        IF finalPosition == 3 THEN
          ;FOLD SPTP P103 Vel=100 % PDAT1 Tool[1]:SMC Base[0] ;%{PE}
          ;FOLD Parameters ;%{h}
          ;Params IlfProvider=kukaroboter.basistech.inlineforms.movement.spline; Kuka.IsGlobalPoint=False; Kuka.PointName=P103; Kuka.BlendingEnabled=False; Kuka.MoveDataPtpName=PDAT1; Kuka.VelocityPtp=100; Kuka.VelocityFieldEnabled=True; Kuka.ColDetectFieldEnabled=True; Kuka.CurrentCDSetIndex=0; Kuka.MovementParameterFieldEnabled=True; IlfCommand=SPTP
          ;ENDFOLD
          SPTP XP103 WITH $VEL_AXIS[1] = SVEL_JOINT(100.0), $TOOL = STOOL2(FP103), $BASE = SBASE(FP103.BASE_NO), $IPO_MODE = SIPO_MODE(FP103.IPO_FRAME), $LOAD = SLOAD(FP103.TOOL_NO), $ACC_AXIS[1] = SACC_JOINT(PPDAT1), $APO = SAPO_PTP(PPDAT1), $GEAR_JERK[1] = SGEAR_JERK(PPDAT1), $COLLMON_TOL_PRO[1] = USE_CM_PRO_VALUES(0)
          ;ENDFOLD
          ;FOLD SLIN P203 Vel=0.1 m/s CPDAT27 Tool[1]:SMC Base[0] ;%{PE}
          ;FOLD Parameters ;%{h}
          ;Params IlfProvider=kukaroboter.basistech.inlineforms.movement.spline; Kuka.IsGlobalPoint=False; Kuka.PointName=P203; Kuka.BlendingEnabled=False; Kuka.MoveDataName=CPDAT27; Kuka.VelocityPath=0.1; Kuka.VelocityFieldEnabled=True; Kuka.ColDetectFieldEnabled=True; Kuka.CurrentCDSetIndex=0; Kuka.MovementParameterFieldEnabled=True; IlfCommand=SLIN
          ;ENDFOLD
          SLIN XP203 WITH $VEL = SVEL_CP(0.1, , LCPDAT27), $TOOL = STOOL2(FP203), $BASE = SBASE(FP203.BASE_NO), $IPO_MODE = SIPO_MODE(FP203.IPO_FRAME), $LOAD = SLOAD(FP203.TOOL_NO), $ACC = SACC_CP(LCPDAT27), $ORI_TYPE = SORI_TYP(LCPDAT27), $APO = SAPO(LCPDAT27), $JERK = SJERK(LCPDAT27), $COLLMON_TOL_PRO[1] = USE_CM_PRO_VALUES(0)
          ;ENDFOLD
          ;FOLD Gripper SET [1]Gripper1 State=[1]ABIERTA Wait 0.2[s] Check with Strategy 1 ;%{PE}
          ;FOLD Parameters Parameters ;%{h}
          ;Params IlfProvider=GripperTech.GripperSet;setgripper=1;setstate=1;setcont=nocont;waittime=0.2;errorstrategy=1
          ;ENDFOLD
          GRPg_SetStateAndCheck(1, 1, 0.2, 1)
          ;ENDFOLD
          ;FOLD SLIN P103 Vel=0.1 m/s CPDAT28 Tool[1]:SMC Base[0] ;%{PE}
          ;FOLD Parameters ;%{h}
          ;Params IlfProvider=kukaroboter.basistech.inlineforms.movement.spline; Kuka.IsGlobalPoint=False; Kuka.PointName=P103; Kuka.BlendingEnabled=False; Kuka.MoveDataName=CPDAT28; Kuka.VelocityPath=0.1; Kuka.VelocityFieldEnabled=True; Kuka.ColDetectFieldEnabled=True; Kuka.CurrentCDSetIndex=0; Kuka.MovementParameterFieldEnabled=True; IlfCommand=SLIN
          ;ENDFOLD
          SLIN XP103 WITH $VEL = SVEL_CP(0.1, , LCPDAT28), $TOOL = STOOL2(FP103), $BASE = SBASE(FP103.BASE_NO), $IPO_MODE = SIPO_MODE(FP103.IPO_FRAME), $LOAD = SLOAD(FP103.TOOL_NO), $ACC = SACC_CP(LCPDAT28), $ORI_TYPE = SORI_TYP(LCPDAT28), $APO = SAPO(LCPDAT28), $JERK = SJERK(LCPDAT28), $COLLMON_TOL_PRO[1] = USE_CM_PRO_VALUES(0)
          ;ENDFOLD
          ;FOLD SPTP P600 Vel=100 % PDAT1 Tool[1]:SMC Base[0] ;%{PE}
          ;FOLD Parameters ;%{h}
          ;Params IlfProvider=kukaroboter.basistech.inlineforms.movement.spline; Kuka.IsGlobalPoint=False; Kuka.PointName=P600; Kuka.BlendingEnabled=False; Kuka.MoveDataPtpName=PDAT1; Kuka.VelocityPtp=100; Kuka.VelocityFieldEnabled=True; Kuka.ColDetectFieldEnabled=True; Kuka.CurrentCDSetIndex=0; Kuka.MovementParameterFieldEnabled=True; IlfCommand=SPTP
          ;ENDFOLD
          SPTP XP600 WITH $VEL_AXIS[1] = SVEL_JOINT(100.0), $TOOL = STOOL2(FP600), $BASE = SBASE(FP600.BASE_NO), $IPO_MODE = SIPO_MODE(FP600.IPO_FRAME), $LOAD = SLOAD(FP600.TOOL_NO), $ACC_AXIS[1] = SACC_JOINT(PPDAT1), $APO = SAPO_PTP(PPDAT1), $GEAR_JERK[1] = SGEAR_JERK(PPDAT1), $COLLMON_TOL_PRO[1] = USE_CM_PRO_VALUES(0)
          ;ENDFOLD
          ;FOLD SLIN P601 Vel=0.1 m/s CPDAT27 Tool[1]:SMC Base[0] ;%{PE}
          ;FOLD Parameters ;%{h}
          ;Params IlfProvider=kukaroboter.basistech.inlineforms.movement.spline; Kuka.IsGlobalPoint=False; Kuka.PointName=P601; Kuka.BlendingEnabled=False; Kuka.MoveDataName=CPDAT27; Kuka.VelocityPath=0.1; Kuka.VelocityFieldEnabled=True; Kuka.ColDetectFieldEnabled=True; Kuka.CurrentCDSetIndex=0; Kuka.MovementParameterFieldEnabled=True; IlfCommand=SLIN
          ;ENDFOLD
          SLIN XP601 WITH $VEL = SVEL_CP(0.1, , LCPDAT27), $TOOL = STOOL2(FP601), $BASE = SBASE(FP601.BASE_NO), $IPO_MODE = SIPO_MODE(FP601.IPO_FRAME), $LOAD = SLOAD(FP601.TOOL_NO), $ACC = SACC_CP(LCPDAT27), $ORI_TYPE = SORI_TYP(LCPDAT27), $APO = SAPO(LCPDAT27), $JERK = SJERK(LCPDAT27), $COLLMON_TOL_PRO[1] = USE_CM_PRO_VALUES(0)
          ;ENDFOLD
          ;FOLD SLIN P602 Vel=0.1 m/s CPDAT27 Tool[1]:SMC Base[0] ;%{PE}
          ;FOLD Parameters ;%{h}
          ;Params IlfProvider=kukaroboter.basistech.inlineforms.movement.spline; Kuka.IsGlobalPoint=False; Kuka.PointName=P602; Kuka.BlendingEnabled=False; Kuka.MoveDataName=CPDAT27; Kuka.VelocityPath=0.1; Kuka.VelocityFieldEnabled=True; Kuka.ColDetectFieldEnabled=True; Kuka.CurrentCDSetIndex=0; Kuka.MovementParameterFieldEnabled=True; IlfCommand=SLIN
          ;ENDFOLD
          SLIN XP602 WITH $VEL = SVEL_CP(0.1, , LCPDAT27), $TOOL = STOOL2(FP602), $BASE = SBASE(FP602.BASE_NO), $IPO_MODE = SIPO_MODE(FP602.IPO_FRAME), $LOAD = SLOAD(FP602.TOOL_NO), $ACC = SACC_CP(LCPDAT27), $ORI_TYPE = SORI_TYP(LCPDAT27), $APO = SAPO(LCPDAT27), $JERK = SJERK(LCPDAT27), $COLLMON_TOL_PRO[1] = USE_CM_PRO_VALUES(0)
          ;ENDFOLD
        ENDIF

        IF finalPosition == 4 THEN
          ;FOLD SPTP P104 Vel=100 % PDAT1 Tool[1]:SMC Base[0] ;%{PE}
          ;FOLD Parameters ;%{h}
          ;Params IlfProvider=kukaroboter.basistech.inlineforms.movement.spline; Kuka.IsGlobalPoint=False; Kuka.PointName=P104; Kuka.BlendingEnabled=False; Kuka.MoveDataPtpName=PDAT1; Kuka.VelocityPtp=100; Kuka.VelocityFieldEnabled=True; Kuka.ColDetectFieldEnabled=True; Kuka.CurrentCDSetIndex=0; Kuka.MovementParameterFieldEnabled=True; IlfCommand=SPTP
          ;ENDFOLD
          SPTP XP104 WITH $VEL_AXIS[1] = SVEL_JOINT(100.0), $TOOL = STOOL2(FP104), $BASE = SBASE(FP104.BASE_NO), $IPO_MODE = SIPO_MODE(FP104.IPO_FRAME), $LOAD = SLOAD(FP104.TOOL_NO), $ACC_AXIS[1] = SACC_JOINT(PPDAT1), $APO = SAPO_PTP(PPDAT1), $GEAR_JERK[1] = SGEAR_JERK(PPDAT1), $COLLMON_TOL_PRO[1] = USE_CM_PRO_VALUES(0)
          ;ENDFOLD
          ;FOLD SLIN P204 Vel=0.1 m/s CPDAT27 Tool[1]:SMC Base[0] ;%{PE}
          ;FOLD Parameters ;%{h}
          ;Params IlfProvider=kukaroboter.basistech.inlineforms.movement.spline; Kuka.IsGlobalPoint=False; Kuka.PointName=P204; Kuka.BlendingEnabled=False; Kuka.MoveDataName=CPDAT27; Kuka.VelocityPath=0.1; Kuka.VelocityFieldEnabled=True; Kuka.ColDetectFieldEnabled=True; Kuka.CurrentCDSetIndex=0; Kuka.MovementParameterFieldEnabled=True; IlfCommand=SLIN
          ;ENDFOLD
          SLIN XP204 WITH $VEL = SVEL_CP(0.1, , LCPDAT27), $TOOL = STOOL2(FP204), $BASE = SBASE(FP204.BASE_NO), $IPO_MODE = SIPO_MODE(FP204.IPO_FRAME), $LOAD = SLOAD(FP204.TOOL_NO), $ACC = SACC_CP(LCPDAT27), $ORI_TYPE = SORI_TYP(LCPDAT27), $APO = SAPO(LCPDAT27), $JERK = SJERK(LCPDAT27), $COLLMON_TOL_PRO[1] = USE_CM_PRO_VALUES(0)
          ;ENDFOLD
          ;FOLD Gripper SET [1]Gripper1 State=[1]ABIERTA Wait 0.2[s] Check with Strategy 1 ;%{PE}
          ;FOLD Parameters Parameters ;%{h}
          ;Params IlfProvider=GripperTech.GripperSet;setgripper=1;setstate=1;setcont=nocont;waittime=0.2;errorstrategy=1
          ;ENDFOLD
          GRPg_SetStateAndCheck(1, 1, 0.2, 1)
          ;ENDFOLD
          ;FOLD SLIN P104 Vel=0.1 m/s CPDAT28 Tool[1]:SMC Base[0] ;%{PE}
          ;FOLD Parameters ;%{h}
          ;Params IlfProvider=kukaroboter.basistech.inlineforms.movement.spline; Kuka.IsGlobalPoint=False; Kuka.PointName=P104; Kuka.BlendingEnabled=False; Kuka.MoveDataName=CPDAT28; Kuka.VelocityPath=0.1; Kuka.VelocityFieldEnabled=True; Kuka.ColDetectFieldEnabled=True; Kuka.CurrentCDSetIndex=0; Kuka.MovementParameterFieldEnabled=True; IlfCommand=SLIN
          ;ENDFOLD
          SLIN XP104 WITH $VEL = SVEL_CP(0.1, , LCPDAT28), $TOOL = STOOL2(FP104), $BASE = SBASE(FP104.BASE_NO), $IPO_MODE = SIPO_MODE(FP104.IPO_FRAME), $LOAD = SLOAD(FP104.TOOL_NO), $ACC = SACC_CP(LCPDAT28), $ORI_TYPE = SORI_TYP(LCPDAT28), $APO = SAPO(LCPDAT28), $JERK = SJERK(LCPDAT28), $COLLMON_TOL_PRO[1] = USE_CM_PRO_VALUES(0)
          ;ENDFOLD
          ;FOLD SPTP P600 Vel=100 % PDAT1 Tool[1]:SMC Base[0] ;%{PE}
          ;FOLD Parameters ;%{h}
          ;Params IlfProvider=kukaroboter.basistech.inlineforms.movement.spline; Kuka.IsGlobalPoint=False; Kuka.PointName=P600; Kuka.BlendingEnabled=False; Kuka.MoveDataPtpName=PDAT1; Kuka.VelocityPtp=100; Kuka.VelocityFieldEnabled=True; Kuka.ColDetectFieldEnabled=True; Kuka.CurrentCDSetIndex=0; Kuka.MovementParameterFieldEnabled=True; IlfCommand=SPTP
          ;ENDFOLD
          SPTP XP600 WITH $VEL_AXIS[1] = SVEL_JOINT(100.0), $TOOL = STOOL2(FP600), $BASE = SBASE(FP600.BASE_NO), $IPO_MODE = SIPO_MODE(FP600.IPO_FRAME), $LOAD = SLOAD(FP600.TOOL_NO), $ACC_AXIS[1] = SACC_JOINT(PPDAT1), $APO = SAPO_PTP(PPDAT1), $GEAR_JERK[1] = SGEAR_JERK(PPDAT1), $COLLMON_TOL_PRO[1] = USE_CM_PRO_VALUES(0)
          ;ENDFOLD
          ;FOLD SLIN P601 Vel=0.1 m/s CPDAT27 Tool[1]:SMC Base[0] ;%{PE}
          ;FOLD Parameters ;%{h}
          ;Params IlfProvider=kukaroboter.basistech.inlineforms.movement.spline; Kuka.IsGlobalPoint=False; Kuka.PointName=P601; Kuka.BlendingEnabled=False; Kuka.MoveDataName=CPDAT27; Kuka.VelocityPath=0.1; Kuka.VelocityFieldEnabled=True; Kuka.ColDetectFieldEnabled=True; Kuka.CurrentCDSetIndex=0; Kuka.MovementParameterFieldEnabled=True; IlfCommand=SLIN
          ;ENDFOLD
          SLIN XP601 WITH $VEL = SVEL_CP(0.1, , LCPDAT27), $TOOL = STOOL2(FP601), $BASE = SBASE(FP601.BASE_NO), $IPO_MODE = SIPO_MODE(FP601.IPO_FRAME), $LOAD = SLOAD(FP601.TOOL_NO), $ACC = SACC_CP(LCPDAT27), $ORI_TYPE = SORI_TYP(LCPDAT27), $APO = SAPO(LCPDAT27), $JERK = SJERK(LCPDAT27), $COLLMON_TOL_PRO[1] = USE_CM_PRO_VALUES(0)
          ;ENDFOLD
          ;FOLD SLIN P602 Vel=0.1 m/s CPDAT27 Tool[1]:SMC Base[0] ;%{PE}
          ;FOLD Parameters ;%{h}
          ;Params IlfProvider=kukaroboter.basistech.inlineforms.movement.spline; Kuka.IsGlobalPoint=False; Kuka.PointName=P602; Kuka.BlendingEnabled=False; Kuka.MoveDataName=CPDAT27; Kuka.VelocityPath=0.1; Kuka.VelocityFieldEnabled=True; Kuka.ColDetectFieldEnabled=True; Kuka.CurrentCDSetIndex=0; Kuka.MovementParameterFieldEnabled=True; IlfCommand=SLIN
          ;ENDFOLD
          SLIN XP602 WITH $VEL = SVEL_CP(0.1, , LCPDAT27), $TOOL = STOOL2(FP602), $BASE = SBASE(FP602.BASE_NO), $IPO_MODE = SIPO_MODE(FP602.IPO_FRAME), $LOAD = SLOAD(FP602.TOOL_NO), $ACC = SACC_CP(LCPDAT27), $ORI_TYPE = SORI_TYP(LCPDAT27), $APO = SAPO(LCPDAT27), $JERK = SJERK(LCPDAT27), $COLLMON_TOL_PRO[1] = USE_CM_PRO_VALUES(0)
          ;ENDFOLD
        ENDIF

        IF finalPosition == 5 THEN
          ;FOLD SPTP P105 Vel=100 % PDAT1 Tool[1]:SMC Base[0] ;%{PE}
          ;FOLD Parameters ;%{h}
          ;Params IlfProvider=kukaroboter.basistech.inlineforms.movement.spline; Kuka.IsGlobalPoint=False; Kuka.PointName=P105; Kuka.BlendingEnabled=False; Kuka.MoveDataPtpName=PDAT1; Kuka.VelocityPtp=100; Kuka.VelocityFieldEnabled=True; Kuka.ColDetectFieldEnabled=True; Kuka.CurrentCDSetIndex=0; Kuka.MovementParameterFieldEnabled=True; IlfCommand=SPTP
          ;ENDFOLD
          SPTP XP105 WITH $VEL_AXIS[1] = SVEL_JOINT(100.0), $TOOL = STOOL2(FP105), $BASE = SBASE(FP105.BASE_NO), $IPO_MODE = SIPO_MODE(FP105.IPO_FRAME), $LOAD = SLOAD(FP105.TOOL_NO), $ACC_AXIS[1] = SACC_JOINT(PPDAT1), $APO = SAPO_PTP(PPDAT1), $GEAR_JERK[1] = SGEAR_JERK(PPDAT1), $COLLMON_TOL_PRO[1] = USE_CM_PRO_VALUES(0)
          ;ENDFOLD
          ;FOLD SLIN P205 Vel=0.1 m/s CPDAT27 Tool[1]:SMC Base[0] ;%{PE}
          ;FOLD Parameters ;%{h}
          ;Params IlfProvider=kukaroboter.basistech.inlineforms.movement.spline; Kuka.IsGlobalPoint=False; Kuka.PointName=P205; Kuka.BlendingEnabled=False; Kuka.MoveDataName=CPDAT27; Kuka.VelocityPath=0.1; Kuka.VelocityFieldEnabled=True; Kuka.ColDetectFieldEnabled=True; Kuka.CurrentCDSetIndex=0; Kuka.MovementParameterFieldEnabled=True; IlfCommand=SLIN
          ;ENDFOLD
          SLIN XP205 WITH $VEL = SVEL_CP(0.1, , LCPDAT27), $TOOL = STOOL2(FP205), $BASE = SBASE(FP205.BASE_NO), $IPO_MODE = SIPO_MODE(FP205.IPO_FRAME), $LOAD = SLOAD(FP205.TOOL_NO), $ACC = SACC_CP(LCPDAT27), $ORI_TYPE = SORI_TYP(LCPDAT27), $APO = SAPO(LCPDAT27), $JERK = SJERK(LCPDAT27), $COLLMON_TOL_PRO[1] = USE_CM_PRO_VALUES(0)
          ;ENDFOLD
          ;FOLD Gripper SET [1]Gripper1 State=[1]ABIERTA Wait 0.2[s] Check with Strategy 1 ;%{PE}
          ;FOLD Parameters Parameters ;%{h}
          ;Params IlfProvider=GripperTech.GripperSet;setgripper=1;setstate=1;setcont=nocont;waittime=0.2;errorstrategy=1
          ;ENDFOLD
          GRPg_SetStateAndCheck(1, 1, 0.2, 1)
          ;ENDFOLD
          ;FOLD SLIN P105 Vel=0.1 m/s CPDAT28 Tool[1]:SMC Base[0] ;%{PE}
          ;FOLD Parameters ;%{h}
          ;Params IlfProvider=kukaroboter.basistech.inlineforms.movement.spline; Kuka.IsGlobalPoint=False; Kuka.PointName=P105; Kuka.BlendingEnabled=False; Kuka.MoveDataName=CPDAT28; Kuka.VelocityPath=0.1; Kuka.VelocityFieldEnabled=True; Kuka.ColDetectFieldEnabled=True; Kuka.CurrentCDSetIndex=0; Kuka.MovementParameterFieldEnabled=True; IlfCommand=SLIN
          ;ENDFOLD
          SLIN XP105 WITH $VEL = SVEL_CP(0.1, , LCPDAT28), $TOOL = STOOL2(FP105), $BASE = SBASE(FP105.BASE_NO), $IPO_MODE = SIPO_MODE(FP105.IPO_FRAME), $LOAD = SLOAD(FP105.TOOL_NO), $ACC = SACC_CP(LCPDAT28), $ORI_TYPE = SORI_TYP(LCPDAT28), $APO = SAPO(LCPDAT28), $JERK = SJERK(LCPDAT28), $COLLMON_TOL_PRO[1] = USE_CM_PRO_VALUES(0)
          ;ENDFOLD
          ;FOLD SPTP P600 Vel=100 % PDAT1 Tool[1]:SMC Base[0] ;%{PE}
          ;FOLD Parameters ;%{h}
          ;Params IlfProvider=kukaroboter.basistech.inlineforms.movement.spline; Kuka.IsGlobalPoint=False; Kuka.PointName=P600; Kuka.BlendingEnabled=False; Kuka.MoveDataPtpName=PDAT1; Kuka.VelocityPtp=100; Kuka.VelocityFieldEnabled=True; Kuka.ColDetectFieldEnabled=True; Kuka.CurrentCDSetIndex=0; Kuka.MovementParameterFieldEnabled=True; IlfCommand=SPTP
          ;ENDFOLD
          SPTP XP600 WITH $VEL_AXIS[1] = SVEL_JOINT(100.0), $TOOL = STOOL2(FP600), $BASE = SBASE(FP600.BASE_NO), $IPO_MODE = SIPO_MODE(FP600.IPO_FRAME), $LOAD = SLOAD(FP600.TOOL_NO), $ACC_AXIS[1] = SACC_JOINT(PPDAT1), $APO = SAPO_PTP(PPDAT1), $GEAR_JERK[1] = SGEAR_JERK(PPDAT1), $COLLMON_TOL_PRO[1] = USE_CM_PRO_VALUES(0)
          ;ENDFOLD
          ;FOLD SLIN P601 Vel=0.1 m/s CPDAT27 Tool[1]:SMC Base[0] ;%{PE}
          ;FOLD Parameters ;%{h}
          ;Params IlfProvider=kukaroboter.basistech.inlineforms.movement.spline; Kuka.IsGlobalPoint=False; Kuka.PointName=P601; Kuka.BlendingEnabled=False; Kuka.MoveDataName=CPDAT27; Kuka.VelocityPath=0.1; Kuka.VelocityFieldEnabled=True; Kuka.ColDetectFieldEnabled=True; Kuka.CurrentCDSetIndex=0; Kuka.MovementParameterFieldEnabled=True; IlfCommand=SLIN
          ;ENDFOLD
          SLIN XP601 WITH $VEL = SVEL_CP(0.1, , LCPDAT27), $TOOL = STOOL2(FP601), $BASE = SBASE(FP601.BASE_NO), $IPO_MODE = SIPO_MODE(FP601.IPO_FRAME), $LOAD = SLOAD(FP601.TOOL_NO), $ACC = SACC_CP(LCPDAT27), $ORI_TYPE = SORI_TYP(LCPDAT27), $APO = SAPO(LCPDAT27), $JERK = SJERK(LCPDAT27), $COLLMON_TOL_PRO[1] = USE_CM_PRO_VALUES(0)
          ;ENDFOLD
          ;FOLD SLIN P602 Vel=0.1 m/s CPDAT27 Tool[1]:SMC Base[0] ;%{PE}
          ;FOLD Parameters ;%{h}
          ;Params IlfProvider=kukaroboter.basistech.inlineforms.movement.spline; Kuka.IsGlobalPoint=False; Kuka.PointName=P602; Kuka.BlendingEnabled=False; Kuka.MoveDataName=CPDAT27; Kuka.VelocityPath=0.1; Kuka.VelocityFieldEnabled=True; Kuka.ColDetectFieldEnabled=True; Kuka.CurrentCDSetIndex=0; Kuka.MovementParameterFieldEnabled=True; IlfCommand=SLIN
          ;ENDFOLD
          SLIN XP602 WITH $VEL = SVEL_CP(0.1, , LCPDAT27), $TOOL = STOOL2(FP602), $BASE = SBASE(FP602.BASE_NO), $IPO_MODE = SIPO_MODE(FP602.IPO_FRAME), $LOAD = SLOAD(FP602.TOOL_NO), $ACC = SACC_CP(LCPDAT27), $ORI_TYPE = SORI_TYP(LCPDAT27), $APO = SAPO(LCPDAT27), $JERK = SJERK(LCPDAT27), $COLLMON_TOL_PRO[1] = USE_CM_PRO_VALUES(0)
          ;ENDFOLD
        ENDIF

        IF finalPosition == 6 THEN
          ;FOLD SPTP P106 Vel=100 % PDAT1 Tool[1]:SMC Base[0] ;%{PE}
          ;FOLD Parameters ;%{h}
          ;Params IlfProvider=kukaroboter.basistech.inlineforms.movement.spline; Kuka.IsGlobalPoint=False; Kuka.PointName=P106; Kuka.BlendingEnabled=False; Kuka.MoveDataPtpName=PDAT1; Kuka.VelocityPtp=100; Kuka.VelocityFieldEnabled=True; Kuka.ColDetectFieldEnabled=True; Kuka.CurrentCDSetIndex=0; Kuka.MovementParameterFieldEnabled=True; IlfCommand=SPTP
          ;ENDFOLD
          SPTP XP106 WITH $VEL_AXIS[1] = SVEL_JOINT(100.0), $TOOL = STOOL2(FP106), $BASE = SBASE(FP106.BASE_NO), $IPO_MODE = SIPO_MODE(FP106.IPO_FRAME), $LOAD = SLOAD(FP106.TOOL_NO), $ACC_AXIS[1] = SACC_JOINT(PPDAT1), $APO = SAPO_PTP(PPDAT1), $GEAR_JERK[1] = SGEAR_JERK(PPDAT1), $COLLMON_TOL_PRO[1] = USE_CM_PRO_VALUES(0)
          ;ENDFOLD
          ;FOLD SLIN P206 Vel=0.1 m/s CPDAT27 Tool[1]:SMC Base[0] ;%{PE}
          ;FOLD Parameters ;%{h}
          ;Params IlfProvider=kukaroboter.basistech.inlineforms.movement.spline; Kuka.IsGlobalPoint=False; Kuka.PointName=P206; Kuka.BlendingEnabled=False; Kuka.MoveDataName=CPDAT27; Kuka.VelocityPath=0.1; Kuka.VelocityFieldEnabled=True; Kuka.ColDetectFieldEnabled=True; Kuka.CurrentCDSetIndex=0; Kuka.MovementParameterFieldEnabled=True; IlfCommand=SLIN
          ;ENDFOLD
          SLIN XP206 WITH $VEL = SVEL_CP(0.1, , LCPDAT27), $TOOL = STOOL2(FP206), $BASE = SBASE(FP206.BASE_NO), $IPO_MODE = SIPO_MODE(FP206.IPO_FRAME), $LOAD = SLOAD(FP206.TOOL_NO), $ACC = SACC_CP(LCPDAT27), $ORI_TYPE = SORI_TYP(LCPDAT27), $APO = SAPO(LCPDAT27), $JERK = SJERK(LCPDAT27), $COLLMON_TOL_PRO[1] = USE_CM_PRO_VALUES(0)
          ;ENDFOLD
          ;FOLD Gripper SET [1]Gripper1 State=[1]ABIERTA Wait 0.2[s] Check with Strategy 1 ;%{PE}
          ;FOLD Parameters Parameters ;%{h}
          ;Params IlfProvider=GripperTech.GripperSet;setgripper=1;setstate=1;setcont=nocont;waittime=0.2;errorstrategy=1
          ;ENDFOLD
          GRPg_SetStateAndCheck(1, 1, 0.2, 1)
          ;ENDFOLD
          ;FOLD SLIN P106 Vel=0.1 m/s CPDAT28 Tool[1]:SMC Base[0] ;%{PE}
          ;FOLD Parameters ;%{h}
          ;Params IlfProvider=kukaroboter.basistech.inlineforms.movement.spline; Kuka.IsGlobalPoint=False; Kuka.PointName=P106; Kuka.BlendingEnabled=False; Kuka.MoveDataName=CPDAT28; Kuka.VelocityPath=0.1; Kuka.VelocityFieldEnabled=True; Kuka.ColDetectFieldEnabled=True; Kuka.CurrentCDSetIndex=0; Kuka.MovementParameterFieldEnabled=True; IlfCommand=SLIN
          ;ENDFOLD
          SLIN XP106 WITH $VEL = SVEL_CP(0.1, , LCPDAT28), $TOOL = STOOL2(FP106), $BASE = SBASE(FP106.BASE_NO), $IPO_MODE = SIPO_MODE(FP106.IPO_FRAME), $LOAD = SLOAD(FP106.TOOL_NO), $ACC = SACC_CP(LCPDAT28), $ORI_TYPE = SORI_TYP(LCPDAT28), $APO = SAPO(LCPDAT28), $JERK = SJERK(LCPDAT28), $COLLMON_TOL_PRO[1] = USE_CM_PRO_VALUES(0)
          ;ENDFOLD
          ;FOLD SPTP P600 Vel=100 % PDAT1 Tool[1]:SMC Base[0] ;%{PE}
          ;FOLD Parameters ;%{h}
          ;Params IlfProvider=kukaroboter.basistech.inlineforms.movement.spline; Kuka.IsGlobalPoint=False; Kuka.PointName=P600; Kuka.BlendingEnabled=False; Kuka.MoveDataPtpName=PDAT1; Kuka.VelocityPtp=100; Kuka.VelocityFieldEnabled=True; Kuka.ColDetectFieldEnabled=True; Kuka.CurrentCDSetIndex=0; Kuka.MovementParameterFieldEnabled=True; IlfCommand=SPTP
          ;ENDFOLD
          SPTP XP600 WITH $VEL_AXIS[1] = SVEL_JOINT(100.0), $TOOL = STOOL2(FP600), $BASE = SBASE(FP600.BASE_NO), $IPO_MODE = SIPO_MODE(FP600.IPO_FRAME), $LOAD = SLOAD(FP600.TOOL_NO), $ACC_AXIS[1] = SACC_JOINT(PPDAT1), $APO = SAPO_PTP(PPDAT1), $GEAR_JERK[1] = SGEAR_JERK(PPDAT1), $COLLMON_TOL_PRO[1] = USE_CM_PRO_VALUES(0)
          ;ENDFOLD
          ;FOLD SLIN P601 Vel=0.1 m/s CPDAT27 Tool[1]:SMC Base[0] ;%{PE}
          ;FOLD Parameters ;%{h}
          ;Params IlfProvider=kukaroboter.basistech.inlineforms.movement.spline; Kuka.IsGlobalPoint=False; Kuka.PointName=P601; Kuka.BlendingEnabled=False; Kuka.MoveDataName=CPDAT27; Kuka.VelocityPath=0.1; Kuka.VelocityFieldEnabled=True; Kuka.ColDetectFieldEnabled=True; Kuka.CurrentCDSetIndex=0; Kuka.MovementParameterFieldEnabled=True; IlfCommand=SLIN
          ;ENDFOLD
          SLIN XP601 WITH $VEL = SVEL_CP(0.1, , LCPDAT27), $TOOL = STOOL2(FP601), $BASE = SBASE(FP601.BASE_NO), $IPO_MODE = SIPO_MODE(FP601.IPO_FRAME), $LOAD = SLOAD(FP601.TOOL_NO), $ACC = SACC_CP(LCPDAT27), $ORI_TYPE = SORI_TYP(LCPDAT27), $APO = SAPO(LCPDAT27), $JERK = SJERK(LCPDAT27), $COLLMON_TOL_PRO[1] = USE_CM_PRO_VALUES(0)
          ;ENDFOLD
          ;FOLD SLIN P602 Vel=0.1 m/s CPDAT27 Tool[1]:SMC Base[0] ;%{PE}
          ;FOLD Parameters ;%{h}
          ;Params IlfProvider=kukaroboter.basistech.inlineforms.movement.spline; Kuka.IsGlobalPoint=False; Kuka.PointName=P602; Kuka.BlendingEnabled=False; Kuka.MoveDataName=CPDAT27; Kuka.VelocityPath=0.1; Kuka.VelocityFieldEnabled=True; Kuka.ColDetectFieldEnabled=True; Kuka.CurrentCDSetIndex=0; Kuka.MovementParameterFieldEnabled=True; IlfCommand=SLIN
          ;ENDFOLD
          SLIN XP602 WITH $VEL = SVEL_CP(0.1, , LCPDAT27), $TOOL = STOOL2(FP602), $BASE = SBASE(FP602.BASE_NO), $IPO_MODE = SIPO_MODE(FP602.IPO_FRAME), $LOAD = SLOAD(FP602.TOOL_NO), $ACC = SACC_CP(LCPDAT27), $ORI_TYPE = SORI_TYP(LCPDAT27), $APO = SAPO(LCPDAT27), $JERK = SJERK(LCPDAT27), $COLLMON_TOL_PRO[1] = USE_CM_PRO_VALUES(0)
          ;ENDFOLD
        ENDIF

        IF finalPosition == 7 THEN
          ;FOLD SPTP P107 Vel=100 % PDAT1 Tool[1]:SMC Base[0] ;%{PE}
          ;FOLD Parameters ;%{h}
          ;Params IlfProvider=kukaroboter.basistech.inlineforms.movement.spline; Kuka.IsGlobalPoint=False; Kuka.PointName=P107; Kuka.BlendingEnabled=False; Kuka.MoveDataPtpName=PDAT1; Kuka.VelocityPtp=100; Kuka.VelocityFieldEnabled=True; Kuka.ColDetectFieldEnabled=True; Kuka.CurrentCDSetIndex=0; Kuka.MovementParameterFieldEnabled=True; IlfCommand=SPTP
          ;ENDFOLD
          SPTP XP107 WITH $VEL_AXIS[1] = SVEL_JOINT(100.0), $TOOL = STOOL2(FP107), $BASE = SBASE(FP107.BASE_NO), $IPO_MODE = SIPO_MODE(FP107.IPO_FRAME), $LOAD = SLOAD(FP107.TOOL_NO), $ACC_AXIS[1] = SACC_JOINT(PPDAT1), $APO = SAPO_PTP(PPDAT1), $GEAR_JERK[1] = SGEAR_JERK(PPDAT1), $COLLMON_TOL_PRO[1] = USE_CM_PRO_VALUES(0)
          ;ENDFOLD
          ;FOLD SLIN P207 Vel=0.1 m/s CPDAT27 Tool[1]:SMC Base[0] ;%{PE}
          ;FOLD Parameters ;%{h}
          ;Params IlfProvider=kukaroboter.basistech.inlineforms.movement.spline; Kuka.IsGlobalPoint=False; Kuka.PointName=P207; Kuka.BlendingEnabled=False; Kuka.MoveDataName=CPDAT27; Kuka.VelocityPath=0.1; Kuka.VelocityFieldEnabled=True; Kuka.ColDetectFieldEnabled=True; Kuka.CurrentCDSetIndex=0; Kuka.MovementParameterFieldEnabled=True; IlfCommand=SLIN
          ;ENDFOLD
          SLIN XP207 WITH $VEL = SVEL_CP(0.1, , LCPDAT27), $TOOL = STOOL2(FP207), $BASE = SBASE(FP207.BASE_NO), $IPO_MODE = SIPO_MODE(FP207.IPO_FRAME), $LOAD = SLOAD(FP207.TOOL_NO), $ACC = SACC_CP(LCPDAT27), $ORI_TYPE = SORI_TYP(LCPDAT27), $APO = SAPO(LCPDAT27), $JERK = SJERK(LCPDAT27), $COLLMON_TOL_PRO[1] = USE_CM_PRO_VALUES(0)
          ;ENDFOLD
          ;FOLD Gripper SET [1]Gripper1 State=[1]ABIERTA Wait 0.2[s] Check with Strategy 1 ;%{PE}
          ;FOLD Parameters Parameters ;%{h}
          ;Params IlfProvider=GripperTech.GripperSet;setgripper=1;setstate=1;setcont=nocont;waittime=0.2;errorstrategy=1
          ;ENDFOLD
          GRPg_SetStateAndCheck(1, 1, 0.2, 1)
          ;ENDFOLD
          ;FOLD SLIN P107 Vel=0.1 m/s CPDAT28 Tool[1]:SMC Base[0] ;%{PE}
          ;FOLD Parameters ;%{h}
          ;Params IlfProvider=kukaroboter.basistech.inlineforms.movement.spline; Kuka.IsGlobalPoint=False; Kuka.PointName=P107; Kuka.BlendingEnabled=False; Kuka.MoveDataName=CPDAT28; Kuka.VelocityPath=0.1; Kuka.VelocityFieldEnabled=True; Kuka.ColDetectFieldEnabled=True; Kuka.CurrentCDSetIndex=0; Kuka.MovementParameterFieldEnabled=True; IlfCommand=SLIN
          ;ENDFOLD
          SLIN XP107 WITH $VEL = SVEL_CP(0.1, , LCPDAT28), $TOOL = STOOL2(FP107), $BASE = SBASE(FP107.BASE_NO), $IPO_MODE = SIPO_MODE(FP107.IPO_FRAME), $LOAD = SLOAD(FP107.TOOL_NO), $ACC = SACC_CP(LCPDAT28), $ORI_TYPE = SORI_TYP(LCPDAT28), $APO = SAPO(LCPDAT28), $JERK = SJERK(LCPDAT28), $COLLMON_TOL_PRO[1] = USE_CM_PRO_VALUES(0)
          ;ENDFOLD
          ;FOLD SPTP P600 Vel=100 % PDAT1 Tool[1]:SMC Base[0] ;%{PE}
          ;FOLD Parameters ;%{h}
          ;Params IlfProvider=kukaroboter.basistech.inlineforms.movement.spline; Kuka.IsGlobalPoint=False; Kuka.PointName=P600; Kuka.BlendingEnabled=False; Kuka.MoveDataPtpName=PDAT1; Kuka.VelocityPtp=100; Kuka.VelocityFieldEnabled=True; Kuka.ColDetectFieldEnabled=True; Kuka.CurrentCDSetIndex=0; Kuka.MovementParameterFieldEnabled=True; IlfCommand=SPTP
          ;ENDFOLD
          SPTP XP600 WITH $VEL_AXIS[1] = SVEL_JOINT(100.0), $TOOL = STOOL2(FP600), $BASE = SBASE(FP600.BASE_NO), $IPO_MODE = SIPO_MODE(FP600.IPO_FRAME), $LOAD = SLOAD(FP600.TOOL_NO), $ACC_AXIS[1] = SACC_JOINT(PPDAT1), $APO = SAPO_PTP(PPDAT1), $GEAR_JERK[1] = SGEAR_JERK(PPDAT1), $COLLMON_TOL_PRO[1] = USE_CM_PRO_VALUES(0)
          ;ENDFOLD
          ;FOLD SLIN P601 Vel=0.1 m/s CPDAT27 Tool[1]:SMC Base[0] ;%{PE}
          ;FOLD Parameters ;%{h}
          ;Params IlfProvider=kukaroboter.basistech.inlineforms.movement.spline; Kuka.IsGlobalPoint=False; Kuka.PointName=P601; Kuka.BlendingEnabled=False; Kuka.MoveDataName=CPDAT27; Kuka.VelocityPath=0.1; Kuka.VelocityFieldEnabled=True; Kuka.ColDetectFieldEnabled=True; Kuka.CurrentCDSetIndex=0; Kuka.MovementParameterFieldEnabled=True; IlfCommand=SLIN
          ;ENDFOLD
          SLIN XP601 WITH $VEL = SVEL_CP(0.1, , LCPDAT27), $TOOL = STOOL2(FP601), $BASE = SBASE(FP601.BASE_NO), $IPO_MODE = SIPO_MODE(FP601.IPO_FRAME), $LOAD = SLOAD(FP601.TOOL_NO), $ACC = SACC_CP(LCPDAT27), $ORI_TYPE = SORI_TYP(LCPDAT27), $APO = SAPO(LCPDAT27), $JERK = SJERK(LCPDAT27), $COLLMON_TOL_PRO[1] = USE_CM_PRO_VALUES(0)
          ;ENDFOLD
          ;FOLD SLIN P602 Vel=0.1 m/s CPDAT27 Tool[1]:SMC Base[0] ;%{PE}
          ;FOLD Parameters ;%{h}
          ;Params IlfProvider=kukaroboter.basistech.inlineforms.movement.spline; Kuka.IsGlobalPoint=False; Kuka.PointName=P602; Kuka.BlendingEnabled=False; Kuka.MoveDataName=CPDAT27; Kuka.VelocityPath=0.1; Kuka.VelocityFieldEnabled=True; Kuka.ColDetectFieldEnabled=True; Kuka.CurrentCDSetIndex=0; Kuka.MovementParameterFieldEnabled=True; IlfCommand=SLIN
          ;ENDFOLD
          SLIN XP602 WITH $VEL = SVEL_CP(0.1, , LCPDAT27), $TOOL = STOOL2(FP602), $BASE = SBASE(FP602.BASE_NO), $IPO_MODE = SIPO_MODE(FP602.IPO_FRAME), $LOAD = SLOAD(FP602.TOOL_NO), $ACC = SACC_CP(LCPDAT27), $ORI_TYPE = SORI_TYP(LCPDAT27), $APO = SAPO(LCPDAT27), $JERK = SJERK(LCPDAT27), $COLLMON_TOL_PRO[1] = USE_CM_PRO_VALUES(0)
          ;ENDFOLD
        ENDIF

        IF finalPosition == 8 THEN
          ;FOLD SPTP P108 Vel=100 % PDAT1 Tool[1]:SMC Base[0] ;%{PE}
          ;FOLD Parameters ;%{h}
          ;Params IlfProvider=kukaroboter.basistech.inlineforms.movement.spline; Kuka.IsGlobalPoint=False; Kuka.PointName=P108; Kuka.BlendingEnabled=False; Kuka.MoveDataPtpName=PDAT1; Kuka.VelocityPtp=100; Kuka.VelocityFieldEnabled=True; Kuka.ColDetectFieldEnabled=True; Kuka.CurrentCDSetIndex=0; Kuka.MovementParameterFieldEnabled=True; IlfCommand=SPTP
          ;ENDFOLD
          SPTP XP108 WITH $VEL_AXIS[1] = SVEL_JOINT(100.0), $TOOL = STOOL2(FP108), $BASE = SBASE(FP108.BASE_NO), $IPO_MODE = SIPO_MODE(FP108.IPO_FRAME), $LOAD = SLOAD(FP108.TOOL_NO), $ACC_AXIS[1] = SACC_JOINT(PPDAT1), $APO = SAPO_PTP(PPDAT1), $GEAR_JERK[1] = SGEAR_JERK(PPDAT1), $COLLMON_TOL_PRO[1] = USE_CM_PRO_VALUES(0)
          ;ENDFOLD
          ;FOLD SLIN P208 Vel=0.1 m/s CPDAT27 Tool[1]:SMC Base[0] ;%{PE}
          ;FOLD Parameters ;%{h}
          ;Params IlfProvider=kukaroboter.basistech.inlineforms.movement.spline; Kuka.IsGlobalPoint=False; Kuka.PointName=P208; Kuka.BlendingEnabled=False; Kuka.MoveDataName=CPDAT27; Kuka.VelocityPath=0.1; Kuka.VelocityFieldEnabled=True; Kuka.ColDetectFieldEnabled=True; Kuka.CurrentCDSetIndex=0; Kuka.MovementParameterFieldEnabled=True; IlfCommand=SLIN
          ;ENDFOLD
          SLIN XP208 WITH $VEL = SVEL_CP(0.1, , LCPDAT27), $TOOL = STOOL2(FP208), $BASE = SBASE(FP208.BASE_NO), $IPO_MODE = SIPO_MODE(FP208.IPO_FRAME), $LOAD = SLOAD(FP208.TOOL_NO), $ACC = SACC_CP(LCPDAT27), $ORI_TYPE = SORI_TYP(LCPDAT27), $APO = SAPO(LCPDAT27), $JERK = SJERK(LCPDAT27), $COLLMON_TOL_PRO[1] = USE_CM_PRO_VALUES(0)
          ;ENDFOLD
          ;FOLD Gripper SET [1]Gripper1 State=[1]ABIERTA Wait 0.2[s] Check with Strategy 1 ;%{PE}
          ;FOLD Parameters Parameters ;%{h}
          ;Params IlfProvider=GripperTech.GripperSet;setgripper=1;setstate=1;setcont=nocont;waittime=0.2;errorstrategy=1
          ;ENDFOLD
          GRPg_SetStateAndCheck(1, 1, 0.2, 1)
          ;ENDFOLD
          ;FOLD SLIN P108 Vel=0.1 m/s CPDAT28 Tool[1]:SMC Base[0] ;%{PE}
          ;FOLD Parameters ;%{h}
          ;Params IlfProvider=kukaroboter.basistech.inlineforms.movement.spline; Kuka.IsGlobalPoint=False; Kuka.PointName=P108; Kuka.BlendingEnabled=False; Kuka.MoveDataName=CPDAT28; Kuka.VelocityPath=0.1; Kuka.VelocityFieldEnabled=True; Kuka.ColDetectFieldEnabled=True; Kuka.CurrentCDSetIndex=0; Kuka.MovementParameterFieldEnabled=True; IlfCommand=SLIN
          ;ENDFOLD
          SLIN XP108 WITH $VEL = SVEL_CP(0.1, , LCPDAT28), $TOOL = STOOL2(FP108), $BASE = SBASE(FP108.BASE_NO), $IPO_MODE = SIPO_MODE(FP108.IPO_FRAME), $LOAD = SLOAD(FP108.TOOL_NO), $ACC = SACC_CP(LCPDAT28), $ORI_TYPE = SORI_TYP(LCPDAT28), $APO = SAPO(LCPDAT28), $JERK = SJERK(LCPDAT28), $COLLMON_TOL_PRO[1] = USE_CM_PRO_VALUES(0)
          ;ENDFOLD
          ;FOLD SPTP P600 Vel=100 % PDAT1 Tool[1]:SMC Base[0] ;%{PE}
          ;FOLD Parameters ;%{h}
          ;Params IlfProvider=kukaroboter.basistech.inlineforms.movement.spline; Kuka.IsGlobalPoint=False; Kuka.PointName=P600; Kuka.BlendingEnabled=False; Kuka.MoveDataPtpName=PDAT1; Kuka.VelocityPtp=100; Kuka.VelocityFieldEnabled=True; Kuka.ColDetectFieldEnabled=True; Kuka.CurrentCDSetIndex=0; Kuka.MovementParameterFieldEnabled=True; IlfCommand=SPTP
          ;ENDFOLD
          SPTP XP600 WITH $VEL_AXIS[1] = SVEL_JOINT(100.0), $TOOL = STOOL2(FP600), $BASE = SBASE(FP600.BASE_NO), $IPO_MODE = SIPO_MODE(FP600.IPO_FRAME), $LOAD = SLOAD(FP600.TOOL_NO), $ACC_AXIS[1] = SACC_JOINT(PPDAT1), $APO = SAPO_PTP(PPDAT1), $GEAR_JERK[1] = SGEAR_JERK(PPDAT1), $COLLMON_TOL_PRO[1] = USE_CM_PRO_VALUES(0)
          ;ENDFOLD
          ;FOLD SLIN P601 Vel=0.1 m/s CPDAT27 Tool[1]:SMC Base[0] ;%{PE}
          ;FOLD Parameters ;%{h}
          ;Params IlfProvider=kukaroboter.basistech.inlineforms.movement.spline; Kuka.IsGlobalPoint=False; Kuka.PointName=P601; Kuka.BlendingEnabled=False; Kuka.MoveDataName=CPDAT27; Kuka.VelocityPath=0.1; Kuka.VelocityFieldEnabled=True; Kuka.ColDetectFieldEnabled=True; Kuka.CurrentCDSetIndex=0; Kuka.MovementParameterFieldEnabled=True; IlfCommand=SLIN
          ;ENDFOLD
          SLIN XP601 WITH $VEL = SVEL_CP(0.1, , LCPDAT27), $TOOL = STOOL2(FP601), $BASE = SBASE(FP601.BASE_NO), $IPO_MODE = SIPO_MODE(FP601.IPO_FRAME), $LOAD = SLOAD(FP601.TOOL_NO), $ACC = SACC_CP(LCPDAT27), $ORI_TYPE = SORI_TYP(LCPDAT27), $APO = SAPO(LCPDAT27), $JERK = SJERK(LCPDAT27), $COLLMON_TOL_PRO[1] = USE_CM_PRO_VALUES(0)
          ;ENDFOLD
          ;FOLD SLIN P602 Vel=0.1 m/s CPDAT27 Tool[1]:SMC Base[0] ;%{PE}
          ;FOLD Parameters ;%{h}
          ;Params IlfProvider=kukaroboter.basistech.inlineforms.movement.spline; Kuka.IsGlobalPoint=False; Kuka.PointName=P602; Kuka.BlendingEnabled=False; Kuka.MoveDataName=CPDAT27; Kuka.VelocityPath=0.1; Kuka.VelocityFieldEnabled=True; Kuka.ColDetectFieldEnabled=True; Kuka.CurrentCDSetIndex=0; Kuka.MovementParameterFieldEnabled=True; IlfCommand=SLIN
          ;ENDFOLD
          SLIN XP602 WITH $VEL = SVEL_CP(0.1, , LCPDAT27), $TOOL = STOOL2(FP602), $BASE = SBASE(FP602.BASE_NO), $IPO_MODE = SIPO_MODE(FP602.IPO_FRAME), $LOAD = SLOAD(FP602.TOOL_NO), $ACC = SACC_CP(LCPDAT27), $ORI_TYPE = SORI_TYP(LCPDAT27), $APO = SAPO(LCPDAT27), $JERK = SJERK(LCPDAT27), $COLLMON_TOL_PRO[1] = USE_CM_PRO_VALUES(0)
          ;ENDFOLD
        ENDIF

        IF finalPosition == 9 THEN
          ;FOLD SPTP P109 Vel=100 % PDAT1 Tool[1]:SMC Base[0] ;%{PE}
          ;FOLD Parameters ;%{h}
          ;Params IlfProvider=kukaroboter.basistech.inlineforms.movement.spline; Kuka.IsGlobalPoint=False; Kuka.PointName=P109; Kuka.BlendingEnabled=False; Kuka.MoveDataPtpName=PDAT1; Kuka.VelocityPtp=100; Kuka.VelocityFieldEnabled=True; Kuka.ColDetectFieldEnabled=True; Kuka.CurrentCDSetIndex=0; Kuka.MovementParameterFieldEnabled=True; IlfCommand=SPTP
          ;ENDFOLD
          SPTP XP109 WITH $VEL_AXIS[1] = SVEL_JOINT(100.0), $TOOL = STOOL2(FP109), $BASE = SBASE(FP109.BASE_NO), $IPO_MODE = SIPO_MODE(FP109.IPO_FRAME), $LOAD = SLOAD(FP109.TOOL_NO), $ACC_AXIS[1] = SACC_JOINT(PPDAT1), $APO = SAPO_PTP(PPDAT1), $GEAR_JERK[1] = SGEAR_JERK(PPDAT1), $COLLMON_TOL_PRO[1] = USE_CM_PRO_VALUES(0)
          ;ENDFOLD
          ;FOLD SLIN P209 Vel=0.1 m/s CPDAT27 Tool[1]:SMC Base[0] ;%{PE}
          ;FOLD Parameters ;%{h}
          ;Params IlfProvider=kukaroboter.basistech.inlineforms.movement.spline; Kuka.IsGlobalPoint=False; Kuka.PointName=P209; Kuka.BlendingEnabled=False; Kuka.MoveDataName=CPDAT27; Kuka.VelocityPath=0.1; Kuka.VelocityFieldEnabled=True; Kuka.ColDetectFieldEnabled=True; Kuka.CurrentCDSetIndex=0; Kuka.MovementParameterFieldEnabled=True; IlfCommand=SLIN
          ;ENDFOLD
          SLIN XP209 WITH $VEL = SVEL_CP(0.1, , LCPDAT27), $TOOL = STOOL2(FP209), $BASE = SBASE(FP209.BASE_NO), $IPO_MODE = SIPO_MODE(FP209.IPO_FRAME), $LOAD = SLOAD(FP209.TOOL_NO), $ACC = SACC_CP(LCPDAT27), $ORI_TYPE = SORI_TYP(LCPDAT27), $APO = SAPO(LCPDAT27), $JERK = SJERK(LCPDAT27), $COLLMON_TOL_PRO[1] = USE_CM_PRO_VALUES(0)
          ;ENDFOLD
          ;FOLD Gripper SET [1]Gripper1 State=[1]ABIERTA Wait 0.2[s] Check with Strategy 1 ;%{PE}
          ;FOLD Parameters Parameters ;%{h}
          ;Params IlfProvider=GripperTech.GripperSet;setgripper=1;setstate=1;setcont=nocont;waittime=0.2;errorstrategy=1
          ;ENDFOLD
          GRPg_SetStateAndCheck(1, 1, 0.2, 1)
          ;ENDFOLD
          ;FOLD SLIN P109 Vel=0.1 m/s CPDAT28 Tool[1]:SMC Base[0] ;%{PE}
          ;FOLD Parameters ;%{h}
          ;Params IlfProvider=kukaroboter.basistech.inlineforms.movement.spline; Kuka.IsGlobalPoint=False; Kuka.PointName=P109; Kuka.BlendingEnabled=False; Kuka.MoveDataName=CPDAT28; Kuka.VelocityPath=0.1; Kuka.VelocityFieldEnabled=True; Kuka.ColDetectFieldEnabled=True; Kuka.CurrentCDSetIndex=0; Kuka.MovementParameterFieldEnabled=True; IlfCommand=SLIN
          ;ENDFOLD
          SLIN XP109 WITH $VEL = SVEL_CP(0.1, , LCPDAT28), $TOOL = STOOL2(FP109), $BASE = SBASE(FP109.BASE_NO), $IPO_MODE = SIPO_MODE(FP109.IPO_FRAME), $LOAD = SLOAD(FP109.TOOL_NO), $ACC = SACC_CP(LCPDAT28), $ORI_TYPE = SORI_TYP(LCPDAT28), $APO = SAPO(LCPDAT28), $JERK = SJERK(LCPDAT28), $COLLMON_TOL_PRO[1] = USE_CM_PRO_VALUES(0)
          ;ENDFOLD
          ;FOLD SPTP P600 Vel=100 % PDAT1 Tool[1]:SMC Base[0] ;%{PE}
          ;FOLD Parameters ;%{h}
          ;Params IlfProvider=kukaroboter.basistech.inlineforms.movement.spline; Kuka.IsGlobalPoint=False; Kuka.PointName=P600; Kuka.BlendingEnabled=False; Kuka.MoveDataPtpName=PDAT1; Kuka.VelocityPtp=100; Kuka.VelocityFieldEnabled=True; Kuka.ColDetectFieldEnabled=True; Kuka.CurrentCDSetIndex=0; Kuka.MovementParameterFieldEnabled=True; IlfCommand=SPTP
          ;ENDFOLD
          SPTP XP600 WITH $VEL_AXIS[1] = SVEL_JOINT(100.0), $TOOL = STOOL2(FP600), $BASE = SBASE(FP600.BASE_NO), $IPO_MODE = SIPO_MODE(FP600.IPO_FRAME), $LOAD = SLOAD(FP600.TOOL_NO), $ACC_AXIS[1] = SACC_JOINT(PPDAT1), $APO = SAPO_PTP(PPDAT1), $GEAR_JERK[1] = SGEAR_JERK(PPDAT1), $COLLMON_TOL_PRO[1] = USE_CM_PRO_VALUES(0)
          ;ENDFOLD
          ;FOLD SLIN P601 Vel=0.1 m/s CPDAT27 Tool[1]:SMC Base[0] ;%{PE}
          ;FOLD Parameters ;%{h}
          ;Params IlfProvider=kukaroboter.basistech.inlineforms.movement.spline; Kuka.IsGlobalPoint=False; Kuka.PointName=P601; Kuka.BlendingEnabled=False; Kuka.MoveDataName=CPDAT27; Kuka.VelocityPath=0.1; Kuka.VelocityFieldEnabled=True; Kuka.ColDetectFieldEnabled=True; Kuka.CurrentCDSetIndex=0; Kuka.MovementParameterFieldEnabled=True; IlfCommand=SLIN
          ;ENDFOLD
          SLIN XP601 WITH $VEL = SVEL_CP(0.1, , LCPDAT27), $TOOL = STOOL2(FP601), $BASE = SBASE(FP601.BASE_NO), $IPO_MODE = SIPO_MODE(FP601.IPO_FRAME), $LOAD = SLOAD(FP601.TOOL_NO), $ACC = SACC_CP(LCPDAT27), $ORI_TYPE = SORI_TYP(LCPDAT27), $APO = SAPO(LCPDAT27), $JERK = SJERK(LCPDAT27), $COLLMON_TOL_PRO[1] = USE_CM_PRO_VALUES(0)
          ;ENDFOLD
          ;FOLD SLIN P602 Vel=0.1 m/s CPDAT27 Tool[1]:SMC Base[0] ;%{PE}
          ;FOLD Parameters ;%{h}
          ;Params IlfProvider=kukaroboter.basistech.inlineforms.movement.spline; Kuka.IsGlobalPoint=False; Kuka.PointName=P602; Kuka.BlendingEnabled=False; Kuka.MoveDataName=CPDAT27; Kuka.VelocityPath=0.1; Kuka.VelocityFieldEnabled=True; Kuka.ColDetectFieldEnabled=True; Kuka.CurrentCDSetIndex=0; Kuka.MovementParameterFieldEnabled=True; IlfCommand=SLIN
          ;ENDFOLD
          SLIN XP602 WITH $VEL = SVEL_CP(0.1, , LCPDAT27), $TOOL = STOOL2(FP602), $BASE = SBASE(FP602.BASE_NO), $IPO_MODE = SIPO_MODE(FP602.IPO_FRAME), $LOAD = SLOAD(FP602.TOOL_NO), $ACC = SACC_CP(LCPDAT27), $ORI_TYPE = SORI_TYP(LCPDAT27), $APO = SAPO(LCPDAT27), $JERK = SJERK(LCPDAT27), $COLLMON_TOL_PRO[1] = USE_CM_PRO_VALUES(0)
          ;ENDFOLD
        ENDIF

        IF finalPosition == 10 THEN
          ;FOLD SPTP P110 Vel=100 % PDAT1 Tool[1]:SMC Base[0] ;%{PE}
          ;FOLD Parameters ;%{h}
          ;Params IlfProvider=kukaroboter.basistech.inlineforms.movement.spline; Kuka.IsGlobalPoint=False; Kuka.PointName=P110; Kuka.BlendingEnabled=False; Kuka.MoveDataPtpName=PDAT1; Kuka.VelocityPtp=100; Kuka.VelocityFieldEnabled=True; Kuka.ColDetectFieldEnabled=True; Kuka.CurrentCDSetIndex=0; Kuka.MovementParameterFieldEnabled=True; IlfCommand=SPTP
          ;ENDFOLD
          SPTP XP110 WITH $VEL_AXIS[1] = SVEL_JOINT(100.0), $TOOL = STOOL2(FP110), $BASE = SBASE(FP110.BASE_NO), $IPO_MODE = SIPO_MODE(FP110.IPO_FRAME), $LOAD = SLOAD(FP110.TOOL_NO), $ACC_AXIS[1] = SACC_JOINT(PPDAT1), $APO = SAPO_PTP(PPDAT1), $GEAR_JERK[1] = SGEAR_JERK(PPDAT1), $COLLMON_TOL_PRO[1] = USE_CM_PRO_VALUES(0)
          ;ENDFOLD
          ;FOLD SLIN P210 Vel=0.1 m/s CPDAT27 Tool[1]:SMC Base[0] ;%{PE}
          ;FOLD Parameters ;%{h}
          ;Params IlfProvider=kukaroboter.basistech.inlineforms.movement.spline; Kuka.IsGlobalPoint=False; Kuka.PointName=P210; Kuka.BlendingEnabled=False; Kuka.MoveDataName=CPDAT27; Kuka.VelocityPath=0.1; Kuka.VelocityFieldEnabled=True; Kuka.ColDetectFieldEnabled=True; Kuka.CurrentCDSetIndex=0; Kuka.MovementParameterFieldEnabled=True; IlfCommand=SLIN
          ;ENDFOLD
          SLIN XP210 WITH $VEL = SVEL_CP(0.1, , LCPDAT27), $TOOL = STOOL2(FP210), $BASE = SBASE(FP210.BASE_NO), $IPO_MODE = SIPO_MODE(FP210.IPO_FRAME), $LOAD = SLOAD(FP210.TOOL_NO), $ACC = SACC_CP(LCPDAT27), $ORI_TYPE = SORI_TYP(LCPDAT27), $APO = SAPO(LCPDAT27), $JERK = SJERK(LCPDAT27), $COLLMON_TOL_PRO[1] = USE_CM_PRO_VALUES(0)
          ;ENDFOLD
          ;FOLD Gripper SET [1]Gripper1 State=[1]ABIERTA Wait 0.2[s] Check with Strategy 1 ;%{PE}
          ;FOLD Parameters Parameters ;%{h}
          ;Params IlfProvider=GripperTech.GripperSet;setgripper=1;setstate=1;setcont=nocont;waittime=0.2;errorstrategy=1
          ;ENDFOLD
          GRPg_SetStateAndCheck(1, 1, 0.2, 1)
          ;ENDFOLD
          ;FOLD SLIN P110 Vel=0.1 m/s CPDAT28 Tool[1]:SMC Base[0] ;%{PE}
          ;FOLD Parameters ;%{h}
          ;Params IlfProvider=kukaroboter.basistech.inlineforms.movement.spline; Kuka.IsGlobalPoint=False; Kuka.PointName=P110; Kuka.BlendingEnabled=False; Kuka.MoveDataName=CPDAT28; Kuka.VelocityPath=0.1; Kuka.VelocityFieldEnabled=True; Kuka.ColDetectFieldEnabled=True; Kuka.CurrentCDSetIndex=0; Kuka.MovementParameterFieldEnabled=True; IlfCommand=SLIN
          ;ENDFOLD
          SLIN XP110 WITH $VEL = SVEL_CP(0.1, , LCPDAT28), $TOOL = STOOL2(FP110), $BASE = SBASE(FP110.BASE_NO), $IPO_MODE = SIPO_MODE(FP110.IPO_FRAME), $LOAD = SLOAD(FP110.TOOL_NO), $ACC = SACC_CP(LCPDAT28), $ORI_TYPE = SORI_TYP(LCPDAT28), $APO = SAPO(LCPDAT28), $JERK = SJERK(LCPDAT28), $COLLMON_TOL_PRO[1] = USE_CM_PRO_VALUES(0)
          ;ENDFOLD
          ;FOLD SPTP P600 Vel=100 % PDAT1 Tool[1]:SMC Base[0] ;%{PE}
          ;FOLD Parameters ;%{h}
          ;Params IlfProvider=kukaroboter.basistech.inlineforms.movement.spline; Kuka.IsGlobalPoint=False; Kuka.PointName=P600; Kuka.BlendingEnabled=False; Kuka.MoveDataPtpName=PDAT1; Kuka.VelocityPtp=100; Kuka.VelocityFieldEnabled=True; Kuka.ColDetectFieldEnabled=True; Kuka.CurrentCDSetIndex=0; Kuka.MovementParameterFieldEnabled=True; IlfCommand=SPTP
          ;ENDFOLD
          SPTP XP600 WITH $VEL_AXIS[1] = SVEL_JOINT(100.0), $TOOL = STOOL2(FP600), $BASE = SBASE(FP600.BASE_NO), $IPO_MODE = SIPO_MODE(FP600.IPO_FRAME), $LOAD = SLOAD(FP600.TOOL_NO), $ACC_AXIS[1] = SACC_JOINT(PPDAT1), $APO = SAPO_PTP(PPDAT1), $GEAR_JERK[1] = SGEAR_JERK(PPDAT1), $COLLMON_TOL_PRO[1] = USE_CM_PRO_VALUES(0)
          ;ENDFOLD
          ;FOLD SLIN P601 Vel=0.1 m/s CPDAT27 Tool[1]:SMC Base[0] ;%{PE}
          ;FOLD Parameters ;%{h}
          ;Params IlfProvider=kukaroboter.basistech.inlineforms.movement.spline; Kuka.IsGlobalPoint=False; Kuka.PointName=P601; Kuka.BlendingEnabled=False; Kuka.MoveDataName=CPDAT27; Kuka.VelocityPath=0.1; Kuka.VelocityFieldEnabled=True; Kuka.ColDetectFieldEnabled=True; Kuka.CurrentCDSetIndex=0; Kuka.MovementParameterFieldEnabled=True; IlfCommand=SLIN
          ;ENDFOLD
          SLIN XP601 WITH $VEL = SVEL_CP(0.1, , LCPDAT27), $TOOL = STOOL2(FP601), $BASE = SBASE(FP601.BASE_NO), $IPO_MODE = SIPO_MODE(FP601.IPO_FRAME), $LOAD = SLOAD(FP601.TOOL_NO), $ACC = SACC_CP(LCPDAT27), $ORI_TYPE = SORI_TYP(LCPDAT27), $APO = SAPO(LCPDAT27), $JERK = SJERK(LCPDAT27), $COLLMON_TOL_PRO[1] = USE_CM_PRO_VALUES(0)
          ;ENDFOLD
          ;FOLD SLIN P602 Vel=0.1 m/s CPDAT27 Tool[1]:SMC Base[0] ;%{PE}
          ;FOLD Parameters ;%{h}
          ;Params IlfProvider=kukaroboter.basistech.inlineforms.movement.spline; Kuka.IsGlobalPoint=False; Kuka.PointName=P602; Kuka.BlendingEnabled=False; Kuka.MoveDataName=CPDAT27; Kuka.VelocityPath=0.1; Kuka.VelocityFieldEnabled=True; Kuka.ColDetectFieldEnabled=True; Kuka.CurrentCDSetIndex=0; Kuka.MovementParameterFieldEnabled=True; IlfCommand=SLIN
          ;ENDFOLD
          SLIN XP602 WITH $VEL = SVEL_CP(0.1, , LCPDAT27), $TOOL = STOOL2(FP602), $BASE = SBASE(FP602.BASE_NO), $IPO_MODE = SIPO_MODE(FP602.IPO_FRAME), $LOAD = SLOAD(FP602.TOOL_NO), $ACC = SACC_CP(LCPDAT27), $ORI_TYPE = SORI_TYP(LCPDAT27), $APO = SAPO(LCPDAT27), $JERK = SJERK(LCPDAT27), $COLLMON_TOL_PRO[1] = USE_CM_PRO_VALUES(0)
          ;ENDFOLD
        ENDIF

        IF finalPosition == 11 THEN
          ;FOLD SPTP P111 Vel=100 % PDAT1 Tool[1]:SMC Base[0] ;%{PE}
          ;FOLD Parameters ;%{h}
          ;Params IlfProvider=kukaroboter.basistech.inlineforms.movement.spline; Kuka.IsGlobalPoint=False; Kuka.PointName=P111; Kuka.BlendingEnabled=False; Kuka.MoveDataPtpName=PDAT1; Kuka.VelocityPtp=100; Kuka.VelocityFieldEnabled=True; Kuka.ColDetectFieldEnabled=True; Kuka.CurrentCDSetIndex=0; Kuka.MovementParameterFieldEnabled=True; IlfCommand=SPTP
          ;ENDFOLD
          SPTP XP111 WITH $VEL_AXIS[1] = SVEL_JOINT(100.0), $TOOL = STOOL2(FP111), $BASE = SBASE(FP111.BASE_NO), $IPO_MODE = SIPO_MODE(FP111.IPO_FRAME), $LOAD = SLOAD(FP111.TOOL_NO), $ACC_AXIS[1] = SACC_JOINT(PPDAT1), $APO = SAPO_PTP(PPDAT1), $GEAR_JERK[1] = SGEAR_JERK(PPDAT1), $COLLMON_TOL_PRO[1] = USE_CM_PRO_VALUES(0)
          ;ENDFOLD
          ;FOLD SLIN P211 Vel=0.1 m/s CPDAT27 Tool[1]:SMC Base[0] ;%{PE}
          ;FOLD Parameters ;%{h}
          ;Params IlfProvider=kukaroboter.basistech.inlineforms.movement.spline; Kuka.IsGlobalPoint=False; Kuka.PointName=P211; Kuka.BlendingEnabled=False; Kuka.MoveDataName=CPDAT27; Kuka.VelocityPath=0.1; Kuka.VelocityFieldEnabled=True; Kuka.ColDetectFieldEnabled=True; Kuka.CurrentCDSetIndex=0; Kuka.MovementParameterFieldEnabled=True; IlfCommand=SLIN
          ;ENDFOLD
          SLIN XP211 WITH $VEL = SVEL_CP(0.1, , LCPDAT27), $TOOL = STOOL2(FP211), $BASE = SBASE(FP211.BASE_NO), $IPO_MODE = SIPO_MODE(FP211.IPO_FRAME), $LOAD = SLOAD(FP211.TOOL_NO), $ACC = SACC_CP(LCPDAT27), $ORI_TYPE = SORI_TYP(LCPDAT27), $APO = SAPO(LCPDAT27), $JERK = SJERK(LCPDAT27), $COLLMON_TOL_PRO[1] = USE_CM_PRO_VALUES(0)
          ;ENDFOLD
          ;FOLD Gripper SET [1]Gripper1 State=[1]ABIERTA Wait 0.2[s] Check with Strategy 1 ;%{PE}
          ;FOLD Parameters Parameters ;%{h}
          ;Params IlfProvider=GripperTech.GripperSet;setgripper=1;setstate=1;setcont=nocont;waittime=0.2;errorstrategy=1
          ;ENDFOLD
          GRPg_SetStateAndCheck(1, 1, 0.2, 1)
          ;ENDFOLD
          ;FOLD SLIN P111 Vel=0.1 m/s CPDAT28 Tool[1]:SMC Base[0] ;%{PE}
          ;FOLD Parameters ;%{h}
          ;Params IlfProvider=kukaroboter.basistech.inlineforms.movement.spline; Kuka.IsGlobalPoint=False; Kuka.PointName=P111; Kuka.BlendingEnabled=False; Kuka.MoveDataName=CPDAT28; Kuka.VelocityPath=0.1; Kuka.VelocityFieldEnabled=True; Kuka.ColDetectFieldEnabled=True; Kuka.CurrentCDSetIndex=0; Kuka.MovementParameterFieldEnabled=True; IlfCommand=SLIN
          ;ENDFOLD
          SLIN XP111 WITH $VEL = SVEL_CP(0.1, , LCPDAT28), $TOOL = STOOL2(FP111), $BASE = SBASE(FP111.BASE_NO), $IPO_MODE = SIPO_MODE(FP111.IPO_FRAME), $LOAD = SLOAD(FP111.TOOL_NO), $ACC = SACC_CP(LCPDAT28), $ORI_TYPE = SORI_TYP(LCPDAT28), $APO = SAPO(LCPDAT28), $JERK = SJERK(LCPDAT28), $COLLMON_TOL_PRO[1] = USE_CM_PRO_VALUES(0)
          ;ENDFOLD
          ;FOLD SPTP P600 Vel=100 % PDAT1 Tool[1]:SMC Base[0] ;%{PE}
          ;FOLD Parameters ;%{h}
          ;Params IlfProvider=kukaroboter.basistech.inlineforms.movement.spline; Kuka.IsGlobalPoint=False; Kuka.PointName=P600; Kuka.BlendingEnabled=False; Kuka.MoveDataPtpName=PDAT1; Kuka.VelocityPtp=100; Kuka.VelocityFieldEnabled=True; Kuka.ColDetectFieldEnabled=True; Kuka.CurrentCDSetIndex=0; Kuka.MovementParameterFieldEnabled=True; IlfCommand=SPTP
          ;ENDFOLD
          SPTP XP600 WITH $VEL_AXIS[1] = SVEL_JOINT(100.0), $TOOL = STOOL2(FP600), $BASE = SBASE(FP600.BASE_NO), $IPO_MODE = SIPO_MODE(FP600.IPO_FRAME), $LOAD = SLOAD(FP600.TOOL_NO), $ACC_AXIS[1] = SACC_JOINT(PPDAT1), $APO = SAPO_PTP(PPDAT1), $GEAR_JERK[1] = SGEAR_JERK(PPDAT1), $COLLMON_TOL_PRO[1] = USE_CM_PRO_VALUES(0)
          ;ENDFOLD
          ;FOLD SLIN P601 Vel=0.1 m/s CPDAT27 Tool[1]:SMC Base[0] ;%{PE}
          ;FOLD Parameters ;%{h}
          ;Params IlfProvider=kukaroboter.basistech.inlineforms.movement.spline; Kuka.IsGlobalPoint=False; Kuka.PointName=P601; Kuka.BlendingEnabled=False; Kuka.MoveDataName=CPDAT27; Kuka.VelocityPath=0.1; Kuka.VelocityFieldEnabled=True; Kuka.ColDetectFieldEnabled=True; Kuka.CurrentCDSetIndex=0; Kuka.MovementParameterFieldEnabled=True; IlfCommand=SLIN
          ;ENDFOLD
          SLIN XP601 WITH $VEL = SVEL_CP(0.1, , LCPDAT27), $TOOL = STOOL2(FP601), $BASE = SBASE(FP601.BASE_NO), $IPO_MODE = SIPO_MODE(FP601.IPO_FRAME), $LOAD = SLOAD(FP601.TOOL_NO), $ACC = SACC_CP(LCPDAT27), $ORI_TYPE = SORI_TYP(LCPDAT27), $APO = SAPO(LCPDAT27), $JERK = SJERK(LCPDAT27), $COLLMON_TOL_PRO[1] = USE_CM_PRO_VALUES(0)
          ;ENDFOLD
          ;FOLD SLIN P602 Vel=0.1 m/s CPDAT27 Tool[1]:SMC Base[0] ;%{PE}
          ;FOLD Parameters ;%{h}
          ;Params IlfProvider=kukaroboter.basistech.inlineforms.movement.spline; Kuka.IsGlobalPoint=False; Kuka.PointName=P602; Kuka.BlendingEnabled=False; Kuka.MoveDataName=CPDAT27; Kuka.VelocityPath=0.1; Kuka.VelocityFieldEnabled=True; Kuka.ColDetectFieldEnabled=True; Kuka.CurrentCDSetIndex=0; Kuka.MovementParameterFieldEnabled=True; IlfCommand=SLIN
          ;ENDFOLD
          SLIN XP602 WITH $VEL = SVEL_CP(0.1, , LCPDAT27), $TOOL = STOOL2(FP602), $BASE = SBASE(FP602.BASE_NO), $IPO_MODE = SIPO_MODE(FP602.IPO_FRAME), $LOAD = SLOAD(FP602.TOOL_NO), $ACC = SACC_CP(LCPDAT27), $ORI_TYPE = SORI_TYP(LCPDAT27), $APO = SAPO(LCPDAT27), $JERK = SJERK(LCPDAT27), $COLLMON_TOL_PRO[1] = USE_CM_PRO_VALUES(0)
          ;ENDFOLD
        ENDIF

        IF finalPosition == 12 THEN
          ;FOLD SPTP P112 Vel=100 % PDAT1 Tool[1]:SMC Base[0] ;%{PE}
          ;FOLD Parameters ;%{h}
          ;Params IlfProvider=kukaroboter.basistech.inlineforms.movement.spline; Kuka.IsGlobalPoint=False; Kuka.PointName=P112; Kuka.BlendingEnabled=False; Kuka.MoveDataPtpName=PDAT1; Kuka.VelocityPtp=100; Kuka.VelocityFieldEnabled=True; Kuka.ColDetectFieldEnabled=True; Kuka.CurrentCDSetIndex=0; Kuka.MovementParameterFieldEnabled=True; IlfCommand=SPTP
          ;ENDFOLD
          SPTP XP112 WITH $VEL_AXIS[1] = SVEL_JOINT(100.0), $TOOL = STOOL2(FP112), $BASE = SBASE(FP112.BASE_NO), $IPO_MODE = SIPO_MODE(FP112.IPO_FRAME), $LOAD = SLOAD(FP112.TOOL_NO), $ACC_AXIS[1] = SACC_JOINT(PPDAT1), $APO = SAPO_PTP(PPDAT1), $GEAR_JERK[1] = SGEAR_JERK(PPDAT1), $COLLMON_TOL_PRO[1] = USE_CM_PRO_VALUES(0)
          ;ENDFOLD
          ;FOLD SLIN P212 Vel=0.1 m/s CPDAT27 Tool[1]:SMC Base[0] ;%{PE}
          ;FOLD Parameters ;%{h}
          ;Params IlfProvider=kukaroboter.basistech.inlineforms.movement.spline; Kuka.IsGlobalPoint=False; Kuka.PointName=P212; Kuka.BlendingEnabled=False; Kuka.MoveDataName=CPDAT27; Kuka.VelocityPath=0.1; Kuka.VelocityFieldEnabled=True; Kuka.ColDetectFieldEnabled=True; Kuka.CurrentCDSetIndex=0; Kuka.MovementParameterFieldEnabled=True; IlfCommand=SLIN
          ;ENDFOLD
          SLIN XP212 WITH $VEL = SVEL_CP(0.1, , LCPDAT27), $TOOL = STOOL2(FP212), $BASE = SBASE(FP212.BASE_NO), $IPO_MODE = SIPO_MODE(FP212.IPO_FRAME), $LOAD = SLOAD(FP212.TOOL_NO), $ACC = SACC_CP(LCPDAT27), $ORI_TYPE = SORI_TYP(LCPDAT27), $APO = SAPO(LCPDAT27), $JERK = SJERK(LCPDAT27), $COLLMON_TOL_PRO[1] = USE_CM_PRO_VALUES(0)
          ;ENDFOLD
          ;FOLD Gripper SET [1]Gripper1 State=[1]ABIERTA Wait 0.2[s] Check with Strategy 1 ;%{PE}
          ;FOLD Parameters Parameters ;%{h}
          ;Params IlfProvider=GripperTech.GripperSet;setgripper=1;setstate=1;setcont=nocont;waittime=0.2;errorstrategy=1
          ;ENDFOLD
          GRPg_SetStateAndCheck(1, 1, 0.2, 1)
          ;ENDFOLD
          ;FOLD SLIN P112 Vel=0.1 m/s CPDAT28 Tool[1]:SMC Base[0] ;%{PE}
          ;FOLD Parameters ;%{h}
          ;Params IlfProvider=kukaroboter.basistech.inlineforms.movement.spline; Kuka.IsGlobalPoint=False; Kuka.PointName=P112; Kuka.BlendingEnabled=False; Kuka.MoveDataName=CPDAT28; Kuka.VelocityPath=0.1; Kuka.VelocityFieldEnabled=True; Kuka.ColDetectFieldEnabled=True; Kuka.CurrentCDSetIndex=0; Kuka.MovementParameterFieldEnabled=True; IlfCommand=SLIN
          ;ENDFOLD
          SLIN XP112 WITH $VEL = SVEL_CP(0.1, , LCPDAT28), $TOOL = STOOL2(FP112), $BASE = SBASE(FP112.BASE_NO), $IPO_MODE = SIPO_MODE(FP112.IPO_FRAME), $LOAD = SLOAD(FP112.TOOL_NO), $ACC = SACC_CP(LCPDAT28), $ORI_TYPE = SORI_TYP(LCPDAT28), $APO = SAPO(LCPDAT28), $JERK = SJERK(LCPDAT28), $COLLMON_TOL_PRO[1] = USE_CM_PRO_VALUES(0)
          ;ENDFOLD
          ;FOLD SPTP P600 Vel=100 % PDAT1 Tool[1]:SMC Base[0] ;%{PE}
          ;FOLD Parameters ;%{h}
          ;Params IlfProvider=kukaroboter.basistech.inlineforms.movement.spline; Kuka.IsGlobalPoint=False; Kuka.PointName=P600; Kuka.BlendingEnabled=False; Kuka.MoveDataPtpName=PDAT1; Kuka.VelocityPtp=100; Kuka.VelocityFieldEnabled=True; Kuka.ColDetectFieldEnabled=True; Kuka.CurrentCDSetIndex=0; Kuka.MovementParameterFieldEnabled=True; IlfCommand=SPTP
          ;ENDFOLD
          SPTP XP600 WITH $VEL_AXIS[1] = SVEL_JOINT(100.0), $TOOL = STOOL2(FP600), $BASE = SBASE(FP600.BASE_NO), $IPO_MODE = SIPO_MODE(FP600.IPO_FRAME), $LOAD = SLOAD(FP600.TOOL_NO), $ACC_AXIS[1] = SACC_JOINT(PPDAT1), $APO = SAPO_PTP(PPDAT1), $GEAR_JERK[1] = SGEAR_JERK(PPDAT1), $COLLMON_TOL_PRO[1] = USE_CM_PRO_VALUES(0)
          ;ENDFOLD
          ;FOLD SLIN P601 Vel=0.1 m/s CPDAT27 Tool[1]:SMC Base[0] ;%{PE}
          ;FOLD Parameters ;%{h}
          ;Params IlfProvider=kukaroboter.basistech.inlineforms.movement.spline; Kuka.IsGlobalPoint=False; Kuka.PointName=P601; Kuka.BlendingEnabled=False; Kuka.MoveDataName=CPDAT27; Kuka.VelocityPath=0.1; Kuka.VelocityFieldEnabled=True; Kuka.ColDetectFieldEnabled=True; Kuka.CurrentCDSetIndex=0; Kuka.MovementParameterFieldEnabled=True; IlfCommand=SLIN
          ;ENDFOLD
          SLIN XP601 WITH $VEL = SVEL_CP(0.1, , LCPDAT27), $TOOL = STOOL2(FP601), $BASE = SBASE(FP601.BASE_NO), $IPO_MODE = SIPO_MODE(FP601.IPO_FRAME), $LOAD = SLOAD(FP601.TOOL_NO), $ACC = SACC_CP(LCPDAT27), $ORI_TYPE = SORI_TYP(LCPDAT27), $APO = SAPO(LCPDAT27), $JERK = SJERK(LCPDAT27), $COLLMON_TOL_PRO[1] = USE_CM_PRO_VALUES(0)
          ;ENDFOLD
          ;FOLD SLIN P602 Vel=0.1 m/s CPDAT27 Tool[1]:SMC Base[0] ;%{PE}
          ;FOLD Parameters ;%{h}
          ;Params IlfProvider=kukaroboter.basistech.inlineforms.movement.spline; Kuka.IsGlobalPoint=False; Kuka.PointName=P602; Kuka.BlendingEnabled=False; Kuka.MoveDataName=CPDAT27; Kuka.VelocityPath=0.1; Kuka.VelocityFieldEnabled=True; Kuka.ColDetectFieldEnabled=True; Kuka.CurrentCDSetIndex=0; Kuka.MovementParameterFieldEnabled=True; IlfCommand=SLIN
          ;ENDFOLD
          SLIN XP602 WITH $VEL = SVEL_CP(0.1, , LCPDAT27), $TOOL = STOOL2(FP602), $BASE = SBASE(FP602.BASE_NO), $IPO_MODE = SIPO_MODE(FP602.IPO_FRAME), $LOAD = SLOAD(FP602.TOOL_NO), $ACC = SACC_CP(LCPDAT27), $ORI_TYPE = SORI_TYP(LCPDAT27), $APO = SAPO(LCPDAT27), $JERK = SJERK(LCPDAT27), $COLLMON_TOL_PRO[1] = USE_CM_PRO_VALUES(0)
          ;ENDFOLD
        ENDIF

